// TIA Portal V20 export
VAR_GLOBAL   // PLC tag table "SS0"
   SS0_Column_Green AT %Q2101.4 : Bool;
   SS0_Column_Yellow AT %Q2101.5 : Bool;
   SS0_Column_Red AT %Q2101.6 : Bool;
   SS0_Column_Buzzer AT %Q2101.7 : Bool;
END_VAR
